INTERFACE ITF_SwitchStation EXTENDS __SYSTEM.IQueryInterface

METHOD SwitchMoveComplete : BOOL
VAR_INPUT
END_VAR
END_METHOD

END_INTERFACE

(* stored: Version 1.1.0.1, ProductVersion 3.1.4024.12
   Itf ITF_SwitchStation: Id {73ec2d68-445f-4e3a-b3c8-be66b3feb03c}
   Method SwitchMoveComplete: Id {41f03ef1-25e8-48d2-815a-2864848a925a} *)
